KUKA KRL program: vornull.src, vornull.dat

--- vornull.src ---
&ACCESS RVP
&REL 3
&COMMENT MECH.NULL-UND VORJUSTAGESTELL.
&PARAM TEMPLATE = C:\KRC\ROBOTER\TEMPLATE\VG_APPLPROG
&PARAM EDITMASK = *
DEF  VORNULL ( )
;FOLD INI;%{PE}%V3.2.0,%MKUKATPBASIS,%CINIT,%VCOMMON,%P
;FOLD BAS INI;%{E}%V3.2.0,%MKUKATPBASIS,%CINIT,%VINIT,%P
GLOBAL INTERRUPT DECL 3 WHEN $STOPMESS==TRUE DO IR_STOPM ( )
INTERRUPT ON 3
BAS (#INITMOV,0 )
;ENDFOLD (BAS INI)
;FOLD GRIPPER INI;%{E}%V3.2.0,%MKUKATPGRIPPER,%CINIT,%VINIT,%P
USER_GRP(0,DUMMY,DUMMY,GDEFAULT)
;ENDFOLD (GRIPPER INI)
;FOLD SPOT INI;%{E}%V3.2.0,%MKUKATPSPOT,%CINIT,%VINIT,%P
USERSPOT(#INIT)
;ENDFOLD (SPOT INI)
;FOLD USER INI;%{E}%V3.2.0,%MKUKATPUSER,%CINIT,%VINIT,%P
;Make your modifications here
;ENDFOLD (USER INI)
;ENDFOLD (INI)
;FOLD ; Anlagenbezeichn:               Stations-Nr:;%{PE}%R 3.2.24,%MKUKATPBASIS,%CCOMMENT,%VNORMAL,%P 2:Anlagenbezeichn:               Stations-Nr:
;ENDFOLD
;FOLD ; Stand / Version:;%{PE}%R 3.2.22,%MKUKATPBASIS,%CCOMMENT,%VNORMAL,%P 2:Stand / Version:
;ENDFOLD
;FOLD ; Name Bearbeiter:;%{PE}%R 3.2.22,%MKUKATPBASIS,%CCOMMENT,%VNORMAL,%P 2:Name Bearbeiter:
;ENDFOLD

;FOLD PTP HOME  Vel= 100 % DEFAULT;%{PE}%R 3.2.24,%MKUKATPBASIS,%CMOVE,%VPTP,%P 1:PTP, 2:HOME, 3:, 5:100, 7:DEFAULT
    $BWDSTART = FALSE
    PDAT_ACT=PDEFAULT
    BAS(#PTP_DAT)
    FDAT_ACT=FHOME
    BAS(#FRAMES)
    BAS(#VEL_PTP,100)
    $H_POS=XHOME
    PTP XHOME
;ENDFOLD

WHILE TRUE
  ;zum Anfahren der Nullstellung Satzzeiger setzen
  HALT
ENDWHILE

;FOLD PTP P1  Vel= 100 % PDEFAULT Tool[0] Base[0];%{PE}%R 3.2.24,%MKUKATPBASIS,%CMOVE,%VPTP,%P 1:PTP, 2:P1, 3:, 5:100, 7:PDEFAULT
$BWDSTART = FALSE
PDAT_ACT=PPDEFAULT
BAS(#PTP_DAT)
FDAT_ACT=FP1
BAS(#FRAMES)
BAS(#VEL_PTP,100)
PTP XP1
;ENDFOLD
;FOLD PTP P2  Vel= 100 % PDEFAULT Tool[0] Base[0];%{PE}%R 3.2.24,%MKUKATPBASIS,%CMOVE,%VPTP,%P 1:PTP, 2:P2, 3:, 5:100, 7:PDEFAULT
$BWDSTART = FALSE
PDAT_ACT=PPDEFAULT
BAS(#PTP_DAT)
FDAT_ACT=FP2
BAS(#FRAMES)
BAS(#VEL_PTP,100)
PTP XP2
;ENDFOLD
;FOLD ; Mechanische Null;%{PE}%R 3.2.24,%MKUKATPBASIS,%CCOMMENT,%VNORMAL,%P 2:Mechanische Null
;ENDFOLD
;FOLD PTP Mechnull  Vel= 100 % PDEFAULT;%{PE}%R 3.2.24,%MKUKATPBASIS,%CMOVE,%VPTP,%P 1:PTP, 2:Mechnull, 3:, 5:100, 7:PDEFAULT
$BWDSTART = FALSE
PDAT_ACT=PPDEFAULT
BAS(#PTP_DAT)
FDAT_ACT=FMechnull
BAS(#FRAMES)
BAS(#VEL_PTP,100)
PTP XMechnull
;ENDFOLD
HALT

;FOLD ; Kerben anfahren IR-Vorjustagestellung;%{PE}%R 3.2.24,%MKUKATPBASIS,%CCOMMENT,%VNORMAL,%P 2:Kerben anfahren IR-Vorjustagestellung
;ENDFOLD
;FOLD PTP Vorjus  Vel= 100 % PDEFAULT;%{PE}%R 3.2.24,%MKUKATPBASIS,%CMOVE,%VPTP,%P 1:PTP, 2:Vorjus, 3:, 5:100, 7:PDEFAULT
$BWDSTART = FALSE
PDAT_ACT=PPDEFAULT
BAS(#PTP_DAT)
FDAT_ACT=FVorjus
BAS(#FRAMES)
BAS(#VEL_PTP,100)
PTP XVorjus
;ENDFOLD
;FOLD ; ------------------------------;%{PE}%R 3.2.24,%MKUKATPBASIS,%CCOMMENT,%VNORMAL,%P 2:------------------------------
;ENDFOLD
;FOLD ; Justage !;%{PE}%R 3.2.24,%MKUKATPBASIS,%CCOMMENT,%VNORMAL,%P 2:Justage !
;ENDFOLD
;FOLD ; ------------------------------;%{PE}%R 3.2.24,%MKUKATPBASIS,%CCOMMENT,%VNORMAL,%P 2:------------------------------
;ENDFOLD
;FOLD ; Nullstellung mit Werkzeug;%{PE}%R 3.2.24,%MKUKATPBASIS,%CCOMMENT,%VNORMAL,%P 2:Nullstellung mit Werkzeug
;ENDFOLD

END

--- vornull.dat ---
&ACCESS RVP
&REL 3
&COMMENT MECH.NULL-UND VORJUSTAGESTELL.
&PARAM TEMPLATE = C:\KRC\ROBOTER\TEMPLATE\VG_APPLPROG
&PARAM EDITMASK = *
DEFDAT  VORNULL

;FOLD EXTERNAL DECLARATIONS;%{PE}%V2.2.2,%MKUKATPBASIS,%CEXT,%VCOMMON,%P
;FOLD BAS EXT;%{PE}%V3.2.0,%MKUKATPBASIS,%CEXT,%VEXT,%P
EXT  BAS (BAS_COMMAND  :IN,REAL  :IN )
DECL INT SUCCESS
;ENDFOLD
;FOLD A10 EXT;%{E}%V3.2.0,%MKUKATPARC,%CEXT,%VEXT,%P
EXT  A10 (A_CMD_T:IN,A_STRT_T:IN,A_WELD_T:IN,A_END_T:IN,INT:IN)
;ENDFOLD
;FOLD A20 EXT;%{E}%V3.2.0,%MKUKATPA20,%CEXT,%VEXT,%P
EXT  A20 (INT  :IN,WELD_ST:IN,WELD_FI:IN,INT:IN)
;ENDFOLD
;FOLD GRIPPER EXT;%{E}%V3.2.0,%MKUKATPGRIPPER,%CEXT,%VEXT,%P
EXT  H50 (INT:IN, INT:IN ,INT:IN ,GRP_TYP:IN)
;ENDFOLD
;FOLD SPOT EXT;%{E}%V3.2.0,%MKUKATPSPOT,%CEXT,%VEXT,%P
EXT  USERSPOT (S_COMMAND  :IN, SPOT_TYPE:IN)
;ENDFOLD
;FOLD TOUCHSENSE EXT;%{E}%V3.2.0,%MKUKATPTS,%CEXT,%VEXT,%P
EXT  H70 (INT  :IN,SRCH_TYP_2  :OUT,E6POS  :IN,SRCH_TYP_3  :IN,SRCH_TYP_2  :IN,SRCH_TYP_2  :IN,SRCH_TYP_2  :IN,SRCH_TYP_2  :IN,SRCH_TYP_2  :IN,INT  :IN )
;ENDFOLD
;FOLD USER EXT;%{}%R2.0.2,%MKUKATPUSER,%CEXT,%VEXT,%P
;Make here your modifictions
;ENDFOLD
;ENDFOLD
E6POS XP1={x 0.0,y 0.0,z 0.0,a 0.0,b 0.0,c 0.0,s 2,t 2,e1 0.0,e2 0.0,e3 0.0,e4 0.0,e5 0.0,e6 0.0}
DECL FDAT FP1={TOOL_NO 0,BASE_NO 0,IPO_FRAME #BASE}
DECL PDAT PPDAT1={VEL 100.0,ACC 100.0,APO_DIST 100.0}
E6POS XP2={x 0.0,y 0.0,z 0.0,a 0.0,b 0.0,c 0.0,s 2,t 2,e1 0.0,e2 0.0,e3 0.0,e4 0.0,e5 0.0,e6 0.0}
DECL FDAT FP2={TOOL_NO 0,BASE_NO 0,IPO_FRAME #BASE}
DECL PDAT PPDAT2={VEL 100.0,ACC 100.0,APO_DIST 100.0}
DECL PDAT PPDEFAULT={VEL 100.0,ACC 100.0,APO_DIST 100.0}
E6AXIS XVORJUS={a1 0.700,a2 -89.0,a3 91.2,a4 6.0,a5 2.5,a6 4.0,e1 0.0,e2 0.0,e3 0.0,e4 0.0,e5 0.0,e6 0.0}
DECL FDAT FVORJUS={TOOL_NO 0,BASE_NO 0,IPO_FRAME #BASE}
;FOLD;{H}
DECL BASIS_SUGG_T LAST_BASIS={POINT1[] "P0                      ",POINT2[] "P0                      ",CP_PARAMS[] "CPDAT0                  ",PTP_PARAMS[] "PDAT0                   ",CONT[] "                        ",CP_VEL[] "2                       ",PTP_VEL[] " 100                    "}
ENDDAT
;ENDFOLD
